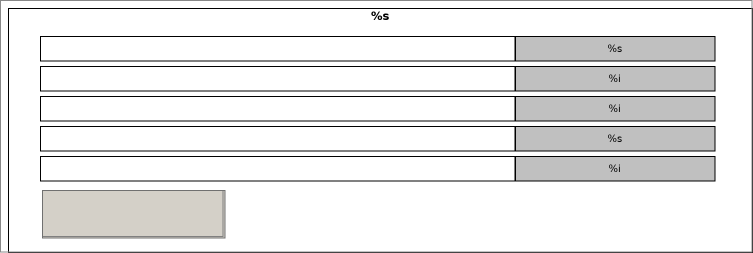
VISUALIZATION VISU_INFO_SUPP_POMPE  // 753x253
VAR_IN_OUT
	COM: BLOCK_RS232_ONBOARD_V4;
END_VAR
    RoundedRectangle (8,8 745x245), "%s", text list: 'TextList_CryoPump', text index: 87
    Rectangle (515,66 200x25), "%i", text variable: COM.Number_Of_Complete_Regen
    Rectangle (40,36 475x25), text list: 'TextList_CryoPump', text index: 47
    Rectangle (40,66 475x25), text list: 'TextList_CryoPump', text index: 48
    Rectangle (40,96 475x25), text list: 'TextList_CryoPump', text index: 49
    Rectangle (40,126 475x25), text list: 'TextList_CryoPump', text index: 50
    Rectangle (40,156 475x25), text list: 'TextList_CryoPump', text index: 51
    Rectangle (515,36 200x25), "%s", text variable: COM.Pump_Serial_Number_affiche
    Rectangle (515,96 200x25), "%i", text variable: COM.Time_Since_Last_Regen
    Rectangle (515,126 200x25), "%s", text variable: COM.SoftwareRevisionLevel
    Rectangle (515,156 200x25), "%i", text variable: COM.ElaspedTime
    Button (42,190 183x48), text list: 'TextList_CryoPump', text index: 88
        OnMouseDown: execute { COM.CO_InfoPompe:=true; }
        OnMouseUp: execute { COM.CO_InfoPompe:=false; }
END_VISUALIZATION

(* stored: Version 1.1.0.1, ProductVersion 3.1.4026.18
   Visu VISU_INFO_SUPP_POMPE: Id {9c6f63c0-39fe-43fb-907d-5fdcda704804} *)
